TYPE UDT_StationReport_RD :
STRUCT
  
alarming : BOOL; // 其它报警中
manualTip : Bool; // 其它手动提示
autoTip : Bool; // 其它自动提示
  
END_STRUCT
END_TYPE

(* stored: Version 1.1.0.1, ProductVersion 3.1.4024.12
   DUT UDT_StationReport_RD: Id {b0bcf481-e378-41d3-9a29-cc72ac9ef5cd} *)
